PROGRAM MAIN
VAR
END_VAR

END_PROGRAM

(* stored: Version 1.1.0.1
   POU MAIN: Id {1850a316-9a69-4bc9-9606-f99d154442e9} *)
